// TwinCAT 3 PLC project PLCStudent
// ProgramVersion: 3.1.4026.21
// libraries:
//   Tc2_Standard, * (Beckhoff Automation GmbH)
//   Tc2_System, * (Beckhoff Automation GmbH)
//   Tc3_Module, * (Beckhoff Automation GmbH)
// project tree:
//   / PlcTask.TcTTO (not stored)
//   POUs/ BLINK.TcPOU, ControlFBD.TcPOU, ControlFBD_Sequence.TcPOU, STATES.TcDUT, MAIN.TcPOU, POUfbd.TcPOU, Sequence.TcPOU
// (motion and I/O tree: see PLC project plcsim)
// real-time tasks:
//   TASK PlcTask: cycle T#30ms, priority 20, ADS port 350
// variable links:
//   PLCSim/PLCSim Instance <-> PLCStudent/PLCStudent Instance
//     PlcTask Inputs/MAIN.ixDrillDown <-> PlcTask Outputs/ControlFBD.qxDrillDown
//     PlcTask Inputs/MAIN.ixDrillUp <-> PlcTask Outputs/ControlFBD.qxDrillUp
//     PlcTask Inputs/MAIN.ixLampEmStopOk <-> PlcTask Outputs/ControlFBD.qxLampEmStopOk
//     PlcTask Inputs/MAIN.ixLampHomePos <-> PlcTask Outputs/ControlFBD.qxLampHomePos
//     PlcTask Inputs/MAIN.ixLampSafetyOk <-> PlcTask Outputs/ControlFBD.qxLampSafetyOk
//     PlcTask Inputs/MAIN.ixLampStarted <-> PlcTask Outputs/ControlFBD.qxLampStarted
//     PlcTask Inputs/MAIN.ixSliderAin <-> PlcTask Outputs/ControlFBD.qxSliderAin
//     PlcTask Inputs/MAIN.ixSliderAout <-> PlcTask Outputs/ControlFBD.qxSliderAout
//     PlcTask Inputs/MAIN.ixSliderBin <-> PlcTask Outputs/ControlFBD.qxSliderBin
//     PlcTask Inputs/MAIN.ixSliderBout <-> PlcTask Outputs/ControlFBD.qxSliderBout
//     PlcTask Outputs/MAIN.qxAuto <-> PlcTask Inputs/ControlFBD.ixAuto
//     PlcTask Outputs/MAIN.qxBtn1EmStopOk <-> PlcTask Inputs/ControlFBD.ixBtn1EmStopOk
//     PlcTask Outputs/MAIN.qxBtn2EmStopOk <-> PlcTask Inputs/ControlFBD.ixBtn2EmStopOk
//     PlcTask Outputs/MAIN.qxBtnAin <-> PlcTask Inputs/ControlFBD.ixBtnAin
//     PlcTask Outputs/MAIN.qxBtnAout <-> PlcTask Inputs/ControlFBD.ixBtnAout
//     PlcTask Outputs/MAIN.qxBtnBin <-> PlcTask Inputs/ControlFBD.ixBtnBin
//     PlcTask Outputs/MAIN.qxBtnBout <-> PlcTask Inputs/ControlFBD.ixBtnBout
//     PlcTask Outputs/MAIN.qxBtnDrillIn <-> PlcTask Inputs/ControlFBD.ixBtnDrillIn
//     PlcTask Outputs/MAIN.qxBtnDrillOut <-> PlcTask Inputs/ControlFBD.ixBtnDrillOut
//     PlcTask Outputs/MAIN.qxBtnReset <-> PlcTask Inputs/ControlFBD.ixBtnReset
//     PlcTask Outputs/MAIN.qxButtonStart <-> PlcTask Inputs/ControlFBD.ixButtonStart
//     PlcTask Outputs/MAIN.qxButtonStop <-> PlcTask Inputs/ControlFBD.ixButtonStop
//     PlcTask Outputs/MAIN.qxDrillDown <-> PlcTask Inputs/ControlFBD.ixDrillDown
//     PlcTask Outputs/MAIN.qxDrillUp <-> PlcTask Inputs/ControlFBD.ixDrillUp
//     PlcTask Outputs/MAIN.qxSafety1StopOk <-> PlcTask Inputs/ControlFBD.ixSafety1StopOk
//     PlcTask Outputs/MAIN.qxSafety2StopOk <-> PlcTask Inputs/ControlFBD.ixSafety2StopOk
//     PlcTask Outputs/MAIN.qxSliderAin <-> PlcTask Inputs/ControlFBD.ixSliderAin
//     PlcTask Outputs/MAIN.qxSliderAout <-> PlcTask Inputs/ControlFBD.ixSliderAout
//     PlcTask Outputs/MAIN.qxSliderBin <-> PlcTask Inputs/ControlFBD.ixSliderBin
//     PlcTask Outputs/MAIN.qxSliderBout <-> PlcTask Inputs/ControlFBD.ixSliderBout

// ---- POUs/STATES.TcDUT
{attribute 'qualified_only'}
{attribute 'strict'}
{attribute 'to_string'}
TYPE STATES :
(
	init,Aout,drillDown,drillUp,Ain,Bout,Bin
);
END_TYPE

// ---- POUs/BLINK.TcPOU
FUNCTION_BLOCK BLINK
VAR_INPUT
	OnTime : TIME;
    OffTime : TIME;
END_VAR

VAR_OUTPUT
    OUT : BOOL;
END_VAR

VAR
    fbTon  : TON;
    fbToff : TON;
END_VAR

fbTon.PT  := OnTime;
fbToff.PT := OffTime;

fbTon.IN := NOT fbToff.Q;
fbTon();

fbToff.IN := fbTon.Q;
fbToff();

Out := fbTon.Q;

END_FUNCTION_BLOCK

// ---- POUs/ControlFBD.TcPOU
PROGRAM ControlFBD
VAR
	qxLampStarted	AT %Q* : BOOL;
	qxSliderAout 	AT %Q* : BOOL; 
	qxSliderAin 	AT %Q* : BOOL; 
	qxSliderBout 	AT %Q* : BOOL; 
	qxSliderBin 	AT %Q* : BOOL; 
	qxDrillDown 	AT %Q* : BOOL;
	qxDrillUp		AT %Q* : BOOL;
	qxLampEmStopOk	AT %Q* : BOOL;
	qxLampSafetyOk  AT %Q* : BOOL;
	qxLampHomePos   AT %Q* : BOOL;
	
	
	ixButtonStart	AT %I* : BOOL;
	ixButtonStop	AT %I* : BOOL;
	ixSliderAout	AT %I* : BOOL;
	ixSliderAin		AT %I* : BOOL;
	ixSliderBout	AT %I* : BOOL;
	ixSliderBin		AT %I* : BOOL;
	ixDrillUp		AT %I* : BOOL;
	ixDrillDown		AT %I* : BOOL;

	ixAuto			AT %I* : BOOL;
	ixBtn1EmStopOk	AT %I* : BOOL;
	ixBtn2EmStopOk	AT %I* : BOOL;	
	ixSafety1StopOk	AT %I* : BOOL;
	ixSafety2StopOk	AT %I* : BOOL;	
	ixBtnReset		AT %I* : BOOL;
	ixBtnAout		AT %I* : BOOL;
	ixBtnAin		AT %I* : BOOL;
	ixBtnBout		AT %I* : BOOL;
	ixBtnBin		AT %I* : BOOL;
	ixBtnDrillOut	AT %I* : BOOL;
	ixBtnDrillIn	AT %I* : BOOL;
    
	mxEmStopReady: BOOL;
	mxEmStopOk: BOOL;
	fbBlink : BLINK;
    mxBlink : BOOL;
	mxSafetyReady: BOOL;
	mxSafetyStopOk: BOOL;
	mxManRunOk: BOOL;
	mxAutoModeReady: BOOL;
	mxCycleStopActivated: BOOL;
	mxAutoRunOk: BOOL;
	BLINK_0: BLINK;
	mxCycleStop: BOOL;
END_VAR
VAR_INPUT
	mxAutoAout: BOOL;
	mxAutoAin: BOOL;
	mxAutoDrillOut: BOOL;
	mxAutoDrillUp: BOOL;
	mxAutoBin: BOOL;
	mxAutoBout: BOOL;
	mxAutoDrillDown: BOOL;
END_VAR

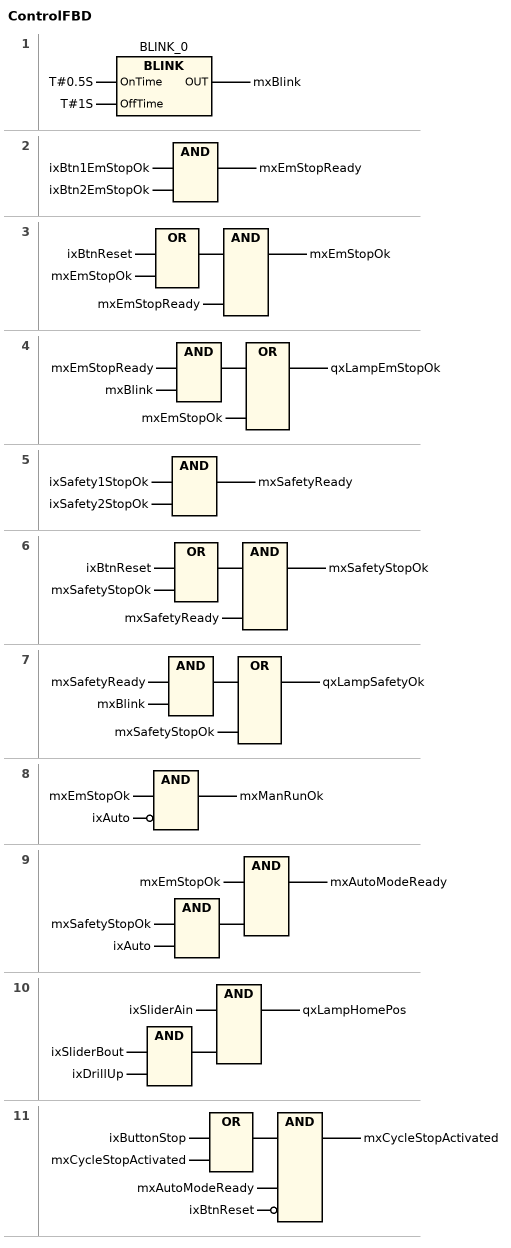
// NETWORK 1
BLINK_0(OnTime := T#0.5S, OffTime := T#1S); // BLINK
mxBlink := BLINK_0.OUT;

// NETWORK 2
mxEmStopReady := ixBtn1EmStopOk AND ixBtn2EmStopOk;

// NETWORK 3
mxEmStopOk := (ixBtnReset OR mxEmStopOk) AND mxEmStopReady;

// NETWORK 4
qxLampEmStopOk := mxEmStopReady AND mxBlink OR mxEmStopOk;

// NETWORK 5
mxSafetyReady := ixSafety1StopOk AND ixSafety2StopOk;

// NETWORK 6
mxSafetyStopOk := (ixBtnReset OR mxSafetyStopOk) AND mxSafetyReady;

// NETWORK 7
qxLampSafetyOk := mxSafetyReady AND mxBlink OR mxSafetyStopOk;

// NETWORK 8
mxManRunOk := mxEmStopOk AND NOT ixAuto;

// NETWORK 9
mxAutoModeReady := mxEmStopOk AND (mxSafetyStopOk AND ixAuto);

// NETWORK 10
qxLampHomePos := ixSliderAin AND (ixSliderBout AND ixDrillUp);

// NETWORK 11
mxCycleStopActivated := (ixButtonStop OR mxCycleStopActivated) AND mxAutoModeReady AND NOT ixBtnReset;

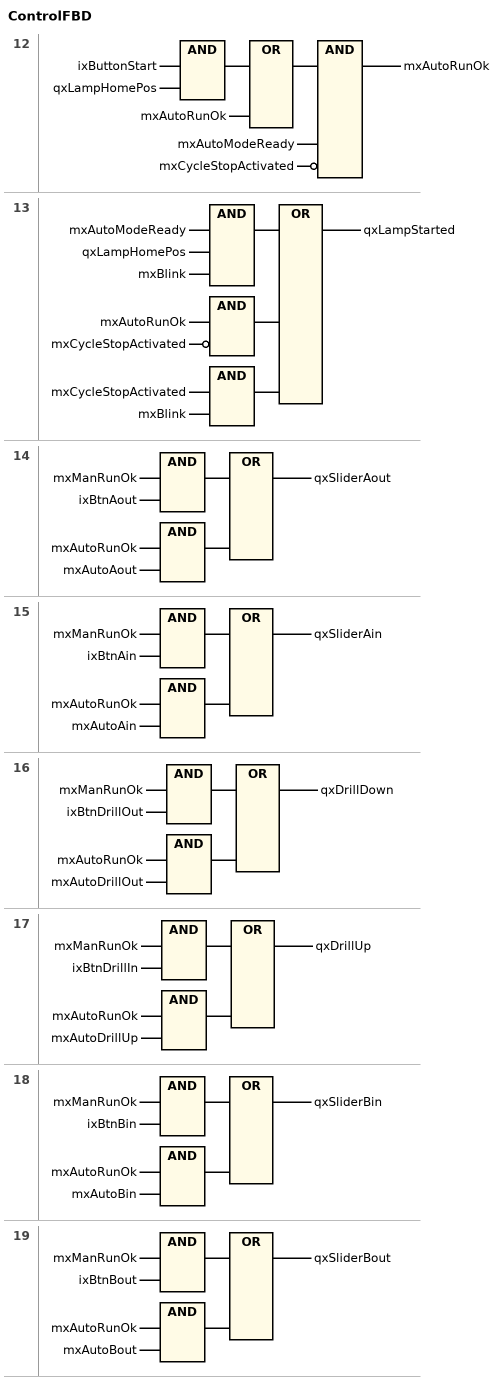
// NETWORK 12
mxAutoRunOk := (ixButtonStart AND qxLampHomePos OR mxAutoRunOk) AND mxAutoModeReady AND NOT mxCycleStopActivated;

// NETWORK 13
qxLampStarted := mxAutoModeReady AND qxLampHomePos AND mxBlink OR mxAutoRunOk AND NOT mxCycleStopActivated OR mxCycleStopActivated AND mxBlink;

// NETWORK 14
qxSliderAout := mxManRunOk AND ixBtnAout OR mxAutoRunOk AND mxAutoAout;

// NETWORK 15
qxSliderAin := mxManRunOk AND ixBtnAin OR mxAutoRunOk AND mxAutoAin;

// NETWORK 16
qxDrillDown := mxManRunOk AND ixBtnDrillOut OR mxAutoRunOk AND mxAutoDrillOut;

// NETWORK 17
qxDrillUp := mxManRunOk AND ixBtnDrillIn OR mxAutoRunOk AND mxAutoDrillUp;

// NETWORK 18
qxSliderBin := mxManRunOk AND ixBtnBin OR mxAutoRunOk AND mxAutoBin;

// NETWORK 19
qxSliderBout := mxManRunOk AND ixBtnBout OR mxAutoRunOk AND mxAutoBout;

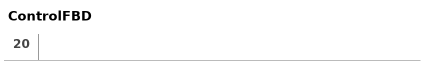
// NETWORK 20

END_PROGRAM

// ---- POUs/ControlFBD_Sequence.TcPOU
FUNCTION_BLOCK ControlFBD_Sequence
VAR_INPUT
	 mxAutoRunOk     : BOOL;
    mxAutoModeReady : BOOL;
    ixSliderAout    : BOOL;
	ixSliderAin    : BOOL;
    ixDrillDown     : BOOL;
    ixDrillUp       : BOOL;
    ixSliderBout    : BOOL;
    ixSliderBin     : BOOL;
END_VAR
VAR_OUTPUT
	mxAutoAout      : BOOL;
    mxAutoDrillDown : BOOL;
    mxAutoDrillUp   : BOOL;
    mxAutoBout      : BOOL;
    mxAutoBin       : BOOL;
    mxAutoAin       : BOOL;
END_VAR
VAR
	miSeq : STATES := STATES.init;
END_VAR

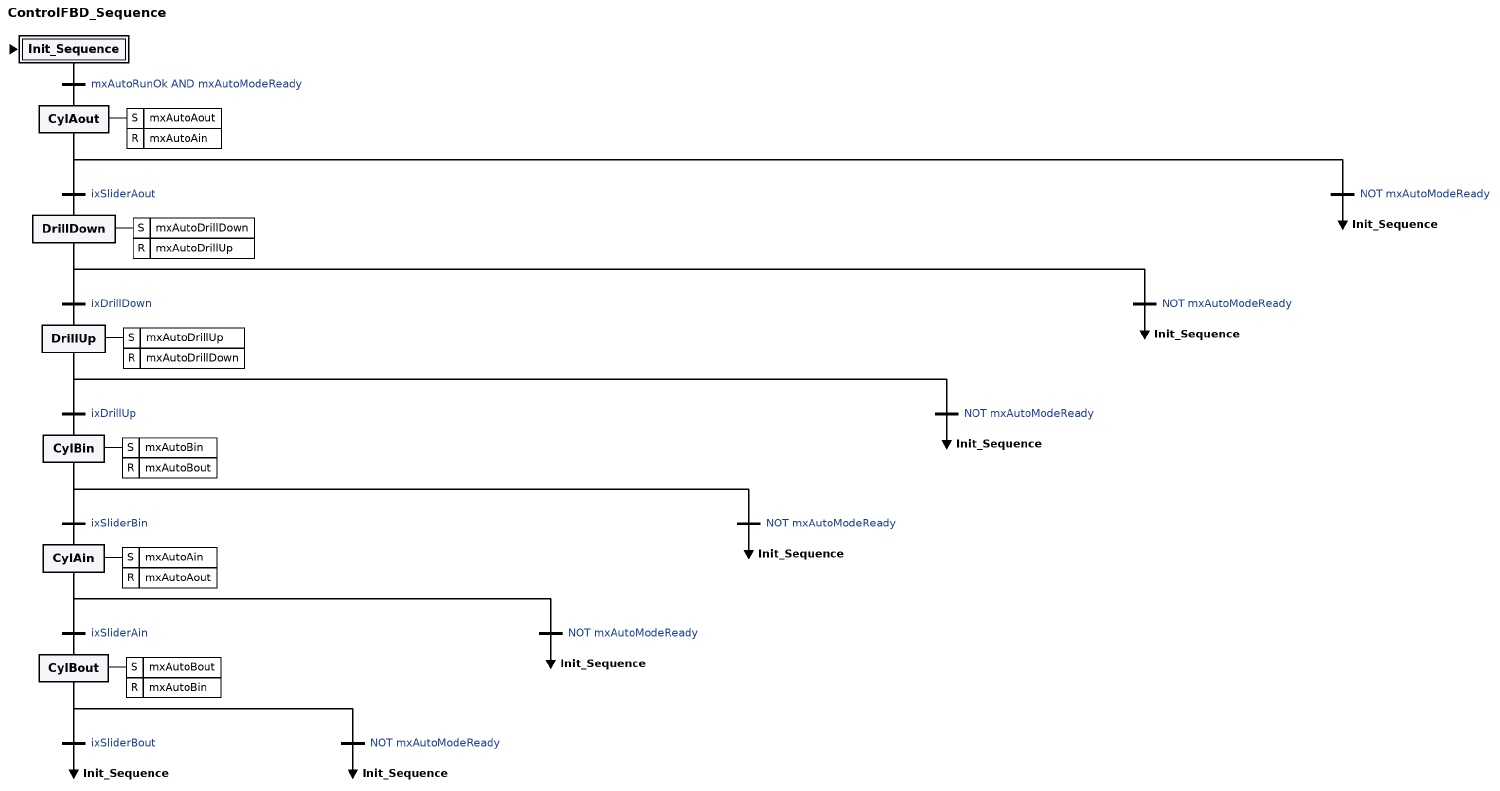
INITIAL_STEP Init_Sequence:
END_STEP
TRANSITION FROM Init_Sequence TO CylAout
    := mxAutoRunOk AND mxAutoModeReady;
END_TRANSITION
STEP CylAout:
    mxAutoAout(S);
    mxAutoAin(R);
END_STEP
TRANSITION FROM CylAout TO DrillDown
    := ixSliderAout;
END_TRANSITION
STEP DrillDown:
    mxAutoDrillDown(S);
    mxAutoDrillUp(R);
END_STEP
TRANSITION FROM DrillDown TO DrillUp
    := ixDrillDown;
END_TRANSITION
STEP DrillUp:
    mxAutoDrillUp(S);
    mxAutoDrillDown(R);
END_STEP
TRANSITION FROM DrillUp TO CylBin
    := ixDrillUp;
END_TRANSITION
STEP CylBin:
    mxAutoBin(S);
    mxAutoBout(R);
END_STEP
TRANSITION FROM CylBin TO CylAin
    := ixSliderBin;
END_TRANSITION
STEP CylAin:
    mxAutoAin(S);
    mxAutoAout(R);
END_STEP
TRANSITION FROM CylAin TO CylBout
    := ixSliderAin;
END_TRANSITION
STEP CylBout:
    mxAutoBout(S);
    mxAutoBin(R);
END_STEP
TRANSITION FROM CylBout TO Init_Sequence
    := ixSliderBout;
END_TRANSITION
TRANSITION FROM CylBout TO Init_Sequence
    := NOT mxAutoModeReady;
END_TRANSITION
TRANSITION FROM CylAin TO Init_Sequence
    := NOT mxAutoModeReady;
END_TRANSITION
TRANSITION FROM CylBin TO Init_Sequence
    := NOT mxAutoModeReady;
END_TRANSITION
TRANSITION FROM DrillUp TO Init_Sequence
    := NOT mxAutoModeReady;
END_TRANSITION
TRANSITION FROM DrillDown TO Init_Sequence
    := NOT mxAutoModeReady;
END_TRANSITION
TRANSITION FROM CylAout TO Init_Sequence
    := NOT mxAutoModeReady;
END_TRANSITION

END_FUNCTION_BLOCK

// ---- POUs/MAIN.TcPOU
PROGRAM MAIN
VAR
	fbSequence : ControlFBD_Sequence;
	fbBlink    : BLINK;
	
	mxAutoRunOk: BOOL;
	mxAutoModeReady: BOOL;
	ixSliderAout: BOOL;
	ixDrillDown: BOOL;
	ixDrillUp: BOOL;
	ixSliderBout: BOOL;
	ixSliderBin: BOOL;
	
	mxAutoAout       : BOOL;
    mxAutoDrillDown: BOOL;
    mxAutoDrillUp    : BOOL;
    mxAutoBout       : BOOL;
    mxAutoBin        : BOOL;
    mxAutoAin        : BOOL;
	
END_VAR

ControlFBD();
(* Auto sequence engine *)
fbSequence(
   mxAutoRunOk     := ControlFBD.mxAutoRunOk,
    mxAutoModeReady := ControlFBD.mxAutoModeReady,
    ixSliderAout    := ControlFBD.ixSliderAout,
    ixDrillDown     := ControlFBD.ixDrillDown,
    ixDrillUp       := ControlFBD.ixDrillUp,
	ixSliderAin    := ControlFBD.ixSliderAin,
    ixSliderBout    := ControlFBD.ixSliderBout,
    ixSliderBin     := ControlFBD.ixSliderBin
);

ControlFBD.mxAutoAout := fbSequence.mxAutoAOut;
ControlFBD.mxAutoAin := fbSequence.mxAutoAIn;
ControlFBD.mxAutoBout := fbSequence.mxAutoBout;
ControlFBD.mxAutoBin := fbSequence.mxAutoBin;
ControlFBD.mxAutoDrillOut := fbSequence.mxAutoDrillDown;
ControlFBD.mxAutoDrillUp := fbSequence.mxAutoDrillUp;

fbBlink(
    OnTime := T#0.5S,
    OffTime := T#1S
);

END_PROGRAM

// ---- POUs/POUfbd.TcPOU
PROGRAM POUfbd
VAR_INPUT
    mxManRunOk : BOOL;
    mxAutoRunOk : BOOL;
    ixBtnAout : BOOL;
    ixBtnAin  : BOOL;
    ixBtnBout : BOOL;
    ixBtnBin  : BOOL;
    ixBtnDrillOut : BOOL;
    ixBtnDrillIn  : BOOL;
END_VAR
VAR_INPUT
    mxAutoAout      : BOOL;
    mxAutoAin       : BOOL;
    mxAutoBout      : BOOL;
    mxAutoBin       : BOOL;
    mxAutoDrillDown : BOOL;
    mxAutoDrillUp   : BOOL;
END_VAR
VAR_OUTPUT
    qxSliderAout : BOOL;
    qxSliderAin  : BOOL;
    qxSliderBout : BOOL;
    qxSliderBin  : BOOL;
    qxDrillDown  : BOOL;
    qxDrillUp    : BOOL;
END_VAR
VAR
	fbBlink : BLINK;
    mxBlink : BOOL;
	mxSumSafetytopReady: BOOL;
	mxSafetyStopOk: BOOL;
	qxLampEmStopOk: BOOL;
	mxEmStopOk: BOOL;
	ixBtnReset: BOOL;
	ixSafety1StopOk: BOOL;
	ixSafety2StopOk: BOOL;
	ixAuto: BOOL;	
	mxAutoModeReady: BOOL;
	ixSliderAin: BOOL;
	ixSlideBout: BOOL;
	ixDrillUp: BOOL;
	qxLampHomePos: BOOL;
	ixButtonStop: BOOL;
	mxCycleStopActivated: BOOL;
	ixButtonStart: BOOL;
	mxCycleStop: BOOL;
	qxLampStarted: BOOL;
	mxAutoDrillOut: BOOL;
END_VAR

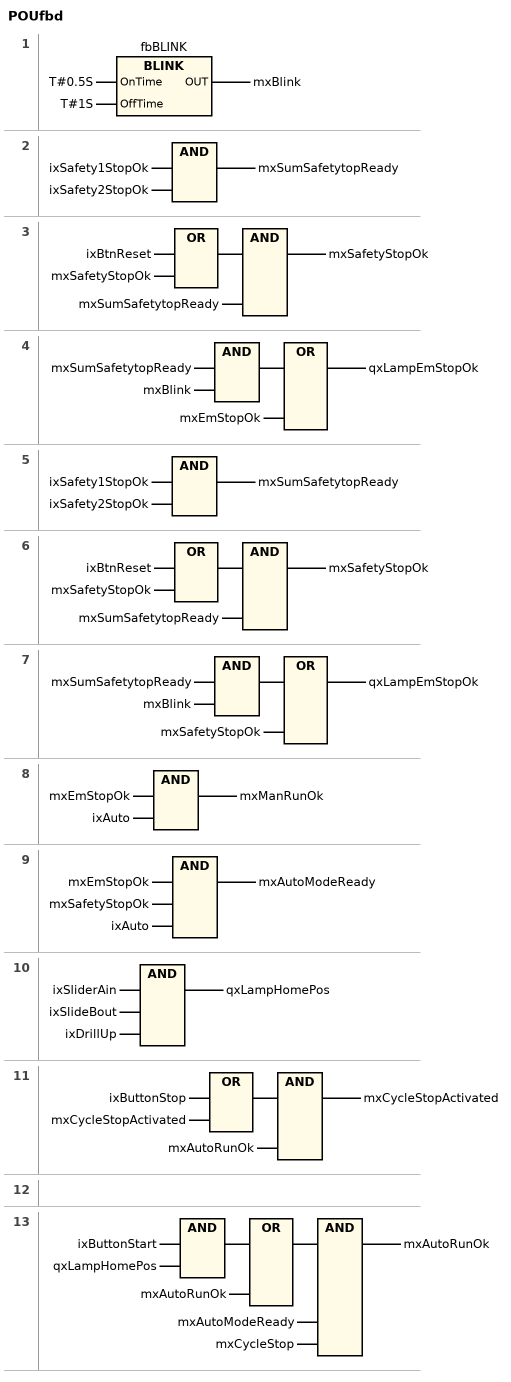
// NETWORK 1
fbBLINK(OnTime := T#0.5S, OffTime := T#1S); // BLINK
mxBlink := fbBLINK.OUT;

// NETWORK 2
mxSumSafetytopReady := ixSafety1StopOk AND ixSafety2StopOk;

// NETWORK 3
mxSafetyStopOk := (ixBtnReset OR mxSafetyStopOk) AND mxSumSafetytopReady;

// NETWORK 4
qxLampEmStopOk := mxSumSafetytopReady AND mxBlink OR mxEmStopOk;

// NETWORK 5
mxSumSafetytopReady := ixSafety1StopOk AND ixSafety2StopOk;

// NETWORK 6
mxSafetyStopOk := (ixBtnReset OR mxSafetyStopOk) AND mxSumSafetytopReady;

// NETWORK 7
qxLampEmStopOk := mxSumSafetytopReady AND mxBlink OR mxSafetyStopOk;

// NETWORK 8
mxManRunOk := mxEmStopOk AND ixAuto;

// NETWORK 9
mxAutoModeReady := mxEmStopOk AND mxSafetyStopOk AND ixAuto;

// NETWORK 10
qxLampHomePos := ixSliderAin AND ixSlideBout AND ixDrillUp;

// NETWORK 11
mxCycleStopActivated := (ixButtonStop OR mxCycleStopActivated) AND mxAutoRunOk;

// NETWORK 12

// NETWORK 13
mxAutoRunOk := (ixButtonStart AND qxLampHomePos OR mxAutoRunOk) AND mxAutoModeReady AND mxCycleStop;

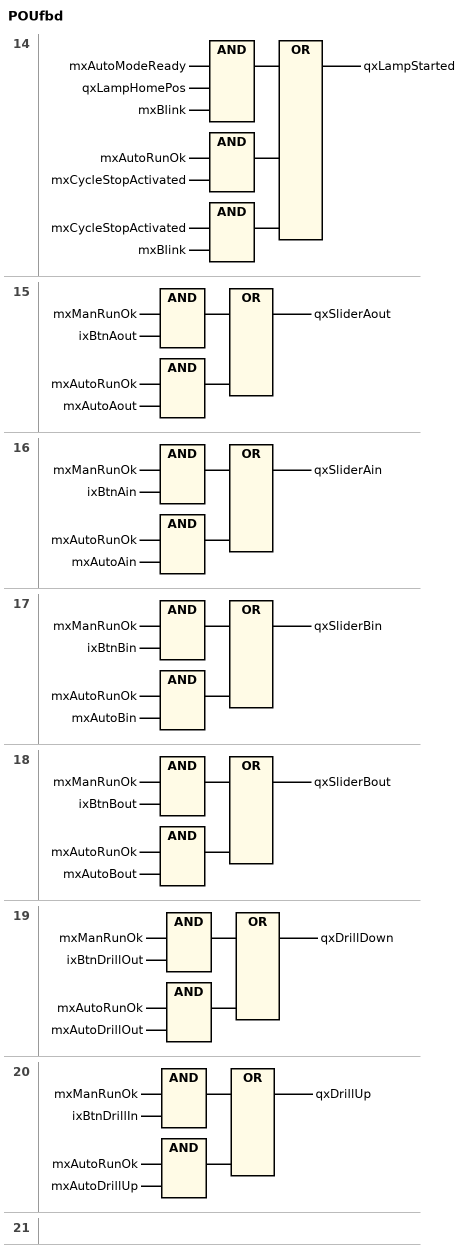
// NETWORK 14
qxLampStarted := mxAutoModeReady AND qxLampHomePos AND mxBlink OR mxAutoRunOk AND mxCycleStopActivated OR mxCycleStopActivated AND mxBlink;

// NETWORK 15
qxSliderAout := mxManRunOk AND ixBtnAout OR mxAutoRunOk AND mxAutoAout;

// NETWORK 16
qxSliderAin := mxManRunOk AND ixBtnAin OR mxAutoRunOk AND mxAutoAin;

// NETWORK 17
qxSliderBin := mxManRunOk AND ixBtnBin OR mxAutoRunOk AND mxAutoBin;

// NETWORK 18
qxSliderBout := mxManRunOk AND ixBtnBout OR mxAutoRunOk AND mxAutoBout;

// NETWORK 19
qxDrillDown := mxManRunOk AND ixBtnDrillOut OR mxAutoRunOk AND mxAutoDrillOut;

// NETWORK 20
qxDrillUp := mxManRunOk AND ixBtnDrillIn OR mxAutoRunOk AND mxAutoDrillUp;

// NETWORK 21

END_PROGRAM

// ---- POUs/Sequence.TcPOU
FUNCTION_BLOCK Sequence
VAR_INPUT
	miSeq: INT;
END_VAR
VAR_OUTPUT
END_VAR
VAR
	mxAutoAout: BOOL;
	mxAutoDrillout: BOOL;
	mxAutoRunOk: BOOL;
	ixSliderAout: BOOL;
	mxAutoBin: BOOL;
	mxAutoBout: BOOL;
	ixDrillDown: BOOL;
	ixDrillUp: BOOL;
	mxAutoAin: BOOL;
	ixSliderBout: BOOL;
	ixSliderBin: BOOL;
	ixSliderAin: BOOL;
END_VAR


CASE miSeq OF

    STATES.init:
        IF mxAutoRunOk THEN
            mxAutoAout := TRUE;
            miSeq := STATES.Aout;
        END_IF

    STATES.Aout:
        IF ixSliderAout THEN
            mxAutoAout := FALSE;
            mxAutoDrillout := TRUE;
            miSeq := STATES.drillDown;
        END_IF

      STATES.drillDown:
          IF ixDrillDown THEN
             mxAutoDrillOut := FALSE;
             miSeq := STATES.drillUp;
        END_IF


      STATES.drillUp:
	     IF ixDrillUp THEN
            mxAutoBout := TRUE;
            miSeq := STATES.Bout;
        END_IF


      STATES.Ain:
           mxAutoAin := TRUE;

        IF ixSliderAin THEN
           mxAutoAin := FALSE;
           mxAutoAout := TRUE;
           miSeq := STATES.Aout;
        END_IF
		
		
      STATES.Bout:
          IF ixSliderBout THEN
             mxAutoBout := FALSE;
             mxAutoBin := TRUE;
             miSeq := STATES.Bin;
         END_IF
	
	  STATES.Bin:
	      IF ixSliderBin THEN
             mxAutoBin := FALSE;
             mxAutoAin := TRUE;
             miSeq := STATES.Ain;
          END_IF
	  	  
END_CASE

END_FUNCTION_BLOCK
